FUNCTION_BLOCK FB_AddAllAxes
VAR_INPUT
	execute: BOOL;
END_VAR
VAR_OUTPUT
	done: BOOL;
	busy: BOOL;
	error: BOOL;
END_VAR
VAR
	fbaddtoaxis: ARRAY[1..grpcnt] OF MC_AddAxisToGroupCA(calltargetOID);
	i: UINT;
END_VAR


done := TRUE;
busy := FALSE;
error := FALSE;

FOR i:=1 TO grpcnt DO
	fbaddtoaxis[i](AxesGroup:=CAgrp, Axis :=grp[i], Execute := execute, IdentInGroup := i-1);

	IF (NOT fbaddtoaxis[i].done) THEN
		done := FALSE;
	END_IF
	IF (fbaddtoaxis[i].busy) THEN
		busy := TRUE;
	END_IF
	IF (fbaddtoaxis[i].Error) THEN
		error := TRUE;
	END_IF
END_FOR

END_FUNCTION_BLOCK

(* stored: Version 1.1.0.1, ProductVersion 3.1.0.25
   POU FB_AddAllAxes: Id {26ec5a14-efc1-4691-b8fc-40bb89bbd235} *)
